# EPICS autosave request: GALIL/iocBoot/iocGALIL-IOC-01/GALIL_01_kinematics.req
file "GALIL_controller_kinematics.req" "P=$(P),CCP=$(CCP)"
